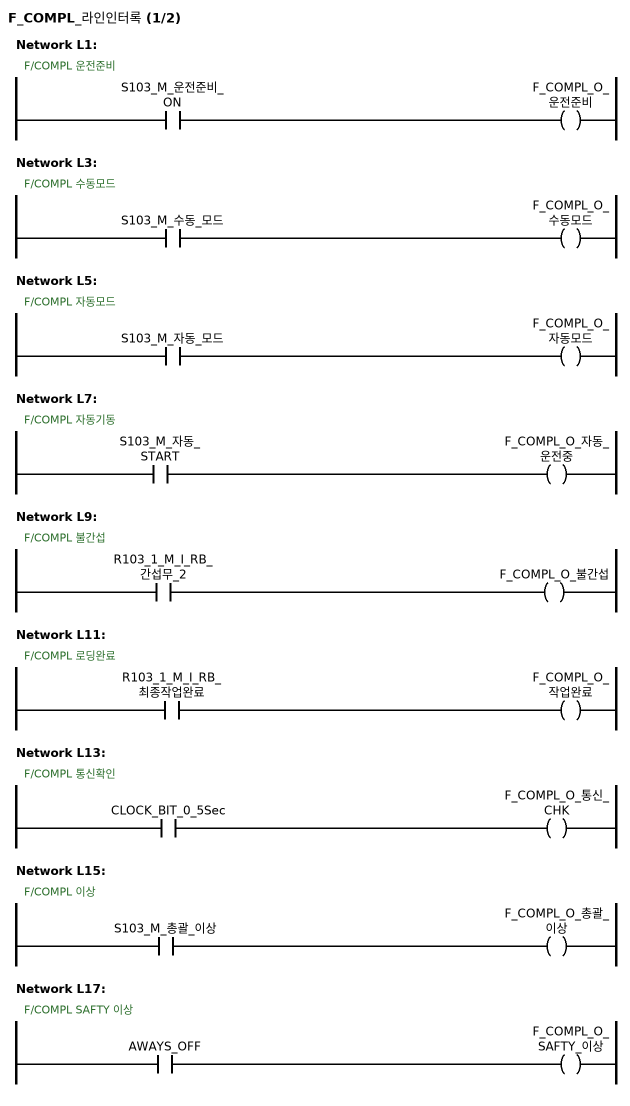
(* [picture p144: F_COMPL_라인인터록 rungs L1-L17] *)
(* F/COMPL 운전준비 *)
(* Rung L1 *)
F_COMPL_O_운전준비 := S103_M_운전준비_ON;
(* F/COMPL 수동모드 *)
(* Rung L3 *)
F_COMPL_O_수동모드 := S103_M_수동_모드;
(* F/COMPL 자동모드 *)
(* Rung L5 *)
F_COMPL_O_자동모드 := S103_M_자동_모드;
(* F/COMPL 자동기동 *)
(* Rung L7 *)
F_COMPL_O_자동_운전중 := S103_M_자동_START;
(* F/COMPL 불간섭 *)
(* Rung L9 *)
F_COMPL_O_불간섭 := R103_1_M_I_RB_간섭무_2;
(* F/COMPL 로딩완료 *)
(* Rung L11 *)
F_COMPL_O_작업완료 := R103_1_M_I_RB_최종작업완료;
(* F/COMPL 통신확인 *)
(* Rung L13 *)
F_COMPL_O_통신_CHK := CLOCK_BIT_0_5Sec;
(* F/COMPL 이상 *)
(* Rung L15 *)
F_COMPL_O_총괄_이상 := S103_M_총괄_이상;
(* F/COMPL SAFTY 이상 *)
(* Rung L17 *)
F_COMPL_O_SAFTY_이상 := AWAYS_OFF;

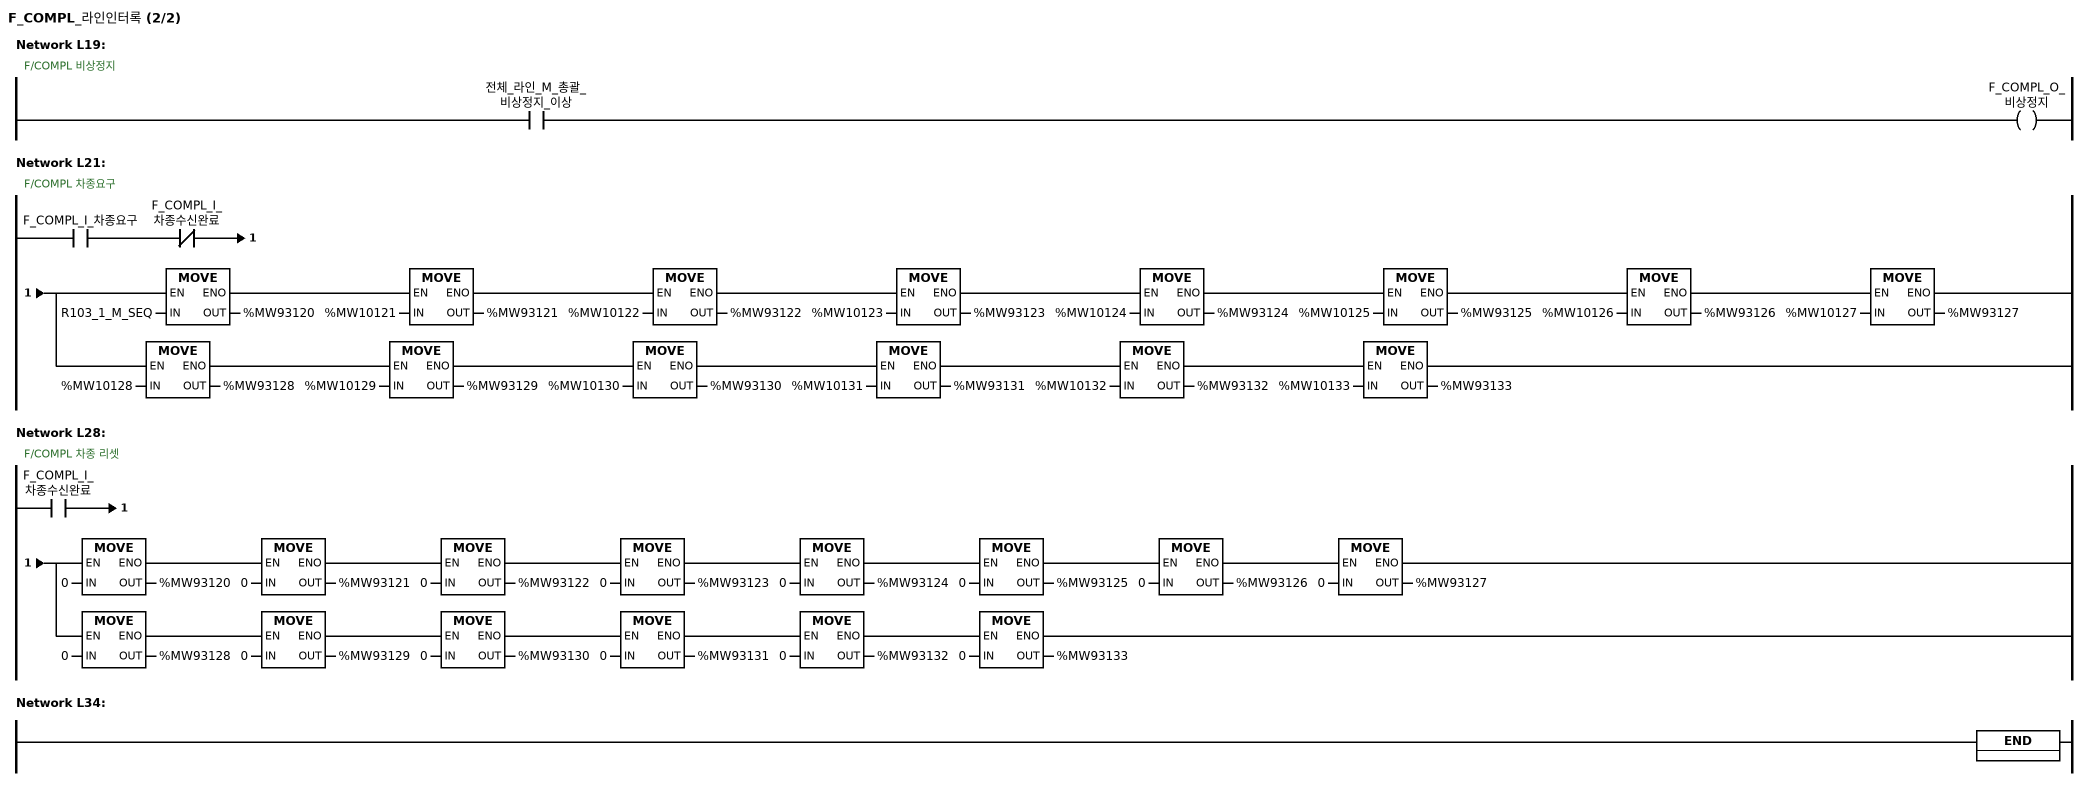
(* F/COMPL 비상정지 *)
(* Rung L19 *)
F_COMPL_O_비상정지 := 전체_라인_M_총괄_비상정지_이상;
(* F/COMPL 차종요구 *)
(* Rung L21 *)
IF F_COMPL_I_차종요구 AND NOT F_COMPL_I_차종수신완료 THEN
    %MW93120 := R103_1_M_SEQ;
    %MW93121 := %MW10121;
    %MW93122 := %MW10122;
    %MW93123 := %MW10123;
    %MW93124 := %MW10124;
    %MW93125 := %MW10125;
    %MW93126 := %MW10126;
    %MW93127 := %MW10127;
    %MW93128 := %MW10128;
    %MW93129 := %MW10129;
    %MW93130 := %MW10130;
    %MW93131 := %MW10131;
    %MW93132 := %MW10132;
    %MW93133 := %MW10133;
END_IF;
(* F/COMPL 차종 리셋 *)
(* Rung L28 *)
IF F_COMPL_I_차종수신완료 THEN
    %MW93120 := 0;
    %MW93121 := 0;
    %MW93122 := 0;
    %MW93123 := 0;
    %MW93124 := 0;
    %MW93125 := 0;
    %MW93126 := 0;
    %MW93127 := 0;
    %MW93128 := 0;
    %MW93129 := 0;
    %MW93130 := 0;
    %MW93131 := 0;
    %MW93132 := 0;
    %MW93133 := 0;
END_IF;
(* Rung L34 *)
END();
END_PROGRAM

PROGRAM 차종전송 (* task: 스캔 프로그램 *)
VAR_EXTERNAL
    AWAYS_OFF : BOOL; (* AT %MW3.0 *)
    AWAYS_ON : BOOL; (* AT %MW3.1 *)
    CARTYPE : ARRAY[0..999] OF WORD; (* AT %MW10000 *) (* CARTYPE *)
    F_COMPL_I_파트_ON : BOOL; (* AT %MW83210.8 *)
    R101_1_1_M_DATA_전송_MEMO : BOOL; (* AT %MW9000.8 *) (* R101_1_1_M_DATA_전송_MEMO *)
    R101_1_1_M_DATA_전송_PLS : BOOL; (* AT %MW9000.9 *) (* R101_1_1_M_DATA_전송_PLS *)
    R101_1_1_M_DATA_전송_완료 : BOOL; (* AT %MW9000.11 *) (* R101_1_1_M_DATA_전송_완료 *)
    R101_1_1_M_STN_차종_ON : BOOL; (* AT %MW1002.2 *)
    R101_1_M_I_RB_2차_작업완료 : BOOL; (* AT %MW20071.3 *)
    R101_1_M_I_RB_원위치 : BOOL; (* AT %MW20070.3 *)
    R101_1_S101_CTYPE_MOVE : FB407_Car_Type_Move_Stn_v1;
    R101_1_S102_CTYPE_MOVE : FB407_Car_Type_Move_Stn_v1;
    R102_1_1_M_DATA_삭제_PLS : BOOL; (* AT %MW9002.0 *) (* R102_1_1_M_DATA_삭제_PLS *)
    R102_1_1_M_DATA_삭제_완료 : BOOL; (* AT %MW9002.2 *) (* R102_1_1_M_DATA_삭제_완료 *)
    R102_1_1_M_DATA_전송_MEMO : BOOL; (* AT %MW9002.8 *) (* R102_1_1_M_DATA_전송_MEMO *)
    R102_1_1_M_DATA_전송_PLS : BOOL; (* AT %MW9002.9 *) (* R102_1_1_M_DATA_전송_PLS *)
    R102_1_1_M_DATA_전송_완료 : BOOL; (* AT %MW9002.11 *) (* R102_1_1_M_DATA_전송_완료 *)
    R102_1_1_M_I_RB_2차_작업완료 : BOOL; (* AT %MW20091.3 *)
    R102_1_1_M_I_RB_원위치 : BOOL; (* AT %MW20090.3 *)
    R102_1_1_M_STN_차종_ON : BOOL; (* AT %MW1502.2 *)
    R102_1_1_S102_CTYPE_MOVE : FB407_Car_Type_Move_Stn_v1;
    R102_1_1_S103_CTYPE_MOVE : FB407_Car_Type_Move_Stn_v1;
    R102_1_CTYPE_CLEAR : FB409_Car_Type_Clear_v1;
    R102_1_M_DATA_전송_MEMO : BOOL; (* AT %MW9004.8 *) (* R102_1_M_DATA_전송_MEMO *)
    R102_1_M_DATA_전송_PLS : BOOL; (* AT %MW9004.9 *) (* R102_1_M_DATA_전송_PLS *)
    R102_1_M_DATA_전송_완료 : BOOL; (* AT %MW9004.11 *) (* R102_1_M_DATA_전송_완료 *)
    R102_1_M_I_RB_1차_작업완료 : BOOL; (* AT %MW20081.2 *)
    R102_1_M_I_RB_2차_작업완료 : BOOL; (* AT %MW20081.3 *)
    R102_1_M_I_RB_원위치 : BOOL; (* AT %MW20080.3 *)
    R102_1_M_STN_차종_NONE : BOOL; (* AT %MW1502.5 *)
    R102_1_M_STN_차종_ON : BOOL; (* AT %MW1502.4 *)
    R102_1_S103_CTYPE_MOVE : FB407_Car_Type_Move_Stn_v1;
    R102_1_S104_CTYPE_MOVE : FB407_Car_Type_Move_Stn_v1;
    R102_2_CTYPE_CLEAR : FB409_Car_Type_Clear_v1;
    R103_1_M_DATA_삭제_PLS : BOOL; (* AT %MW9006.0 *) (* R103_1_M_DATA_삭제_PLS *)
    R103_1_M_DATA_삭제_완료 : BOOL; (* AT %MW9006.2 *) (* R103_1_M_DATA_삭제_완료 *)
    R103_1_M_I_RB_1차_작업완료 : BOOL; (* AT %MW20101.2 *)
    R103_1_M_I_RB_2차_작업완료 : BOOL; (* AT %MW20101.3 *)
    R103_1_M_STN_차종_NONE : BOOL; (* AT %MW2002.3 *)
    S101_M_DATA_전송_MEMO : BOOL; (* AT %MW9001.8 *) (* S101_M_DATA_전송_MEMO *)
    S101_M_DATA_전송_PLS : BOOL; (* AT %MW9001.9 *) (* S101_M_DATA_전송_PLS *)
    S101_M_DATA_전송_완료 : BOOL; (* AT %MW9001.11 *) (* S101_M_DATA_전송_완료 *)
    S101_M_STN_DASH_로딩완료 : BOOL; (* AT %MW1001.12 *)
    S101_M_STN_LH_로딩완료 : BOOL; (* AT %MW1001.10 *)
    S101_M_STN_RH_로딩완료 : BOOL; (* AT %MW1001.11 *)
    S101_M_STN_차종_NONE : BOOL; (* AT %MW1002.1 *)
    S101_M_STN_차종_ON : BOOL; (* AT %MW1002.0 *)
    S101_M_공정_APRON_제품감지_OFF : BOOL; (* AT %MW1001.4 *)
    S101_M_공정_APRON_제품감지_ON : BOOL; (* AT %MW1001.3 *)
    S101_M_공정_DASH_제품감지_OFF : BOOL; (* AT %MW1001.6 *)
    S101_M_작업_완료 : BOOL; (* AT %MW1001.0 *)
    S101_R102_2_CTYPE_MOVE : FB407_Car_Type_Move_Stn_v1;
    S101_R102_3_CTYPE_MOVE : FB407_Car_Type_Move_Stn_v1;
    S102_M_DATA_전송_MEMO : BOOL; (* AT %MW9003.8 *) (* S102_M_DATA_전송_MEMO *)
    S102_M_DATA_전송_PLS : BOOL; (* AT %MW9003.9 *) (* S102_M_DATA_전송_PLS *)
    S102_M_DATA_전송_완료 : BOOL; (* AT %MW9003.11 *) (* S102_M_DATA_전송_완료 *)
    S102_M_STN_DASH_로딩완료 : BOOL; (* AT %MW1501.8 *)
    S102_M_STN_차종_NONE : BOOL; (* AT %MW1502.1 *)
    S102_M_STN_차종_ON : BOOL; (* AT %MW1502.0 *)
    S102_M_공정_제품감지_OFF : BOOL; (* AT %MW1501.4 *)
    S102_M_공정_제품감지_ON : BOOL; (* AT %MW1501.3 *)
    S102_M_작업_완료 : BOOL; (* AT %MW1501.0 *)
    S102_R102_1_CTYPE_MOVE : FB407_Car_Type_Move_Stn_v1;
    S102_R102_2_CTYPE_MOVE : FB407_Car_Type_Move_Stn_v1;
    S103_M_DATA_전송_MEMO : BOOL; (* AT %MW9005.8 *) (* S103_M_DATA_전송_MEMO *)
    S103_M_DATA_전송_PLS : BOOL; (* AT %MW9005.9 *) (* S103_M_DATA_전송_PLS *)
    S103_M_DATA_전송_완료 : BOOL; (* AT %MW9005.11 *) (* S103_M_DATA_전송_완료 *)
    S103_M_STN_FRT_FLR_로딩완료 : BOOL; (* AT %MW2001.8 *)
    S103_M_STN_차종_NONE : BOOL; (* AT %MW2002.1 *)
    S103_M_STN_차종_ON : BOOL; (* AT %MW2002.0 *)
    S103_M_공정_제품감지_OFF : BOOL; (* AT %MW2001.4 *)
    S103_M_공정_제품감지_ON : BOOL; (* AT %MW2001.3 *)
    S103_M_작업_완료 : BOOL; (* AT %MW2001.0 *)
    S103_R103_1_CTYPE_MOVE : FB407_Car_Type_Move_Stn_v1;
    S103_R103_2_CTYPE_MOVE : FB407_Car_Type_Move_Stn_v1;
END_VAR
VAR
    _e1 : R_TRIG;
    _e2 : R_TRIG;
    _e3 : R_TRIG;
    _e4 : R_TRIG;
    _e5 : R_TRIG;
    _e6 : R_TRIG;
END_VAR

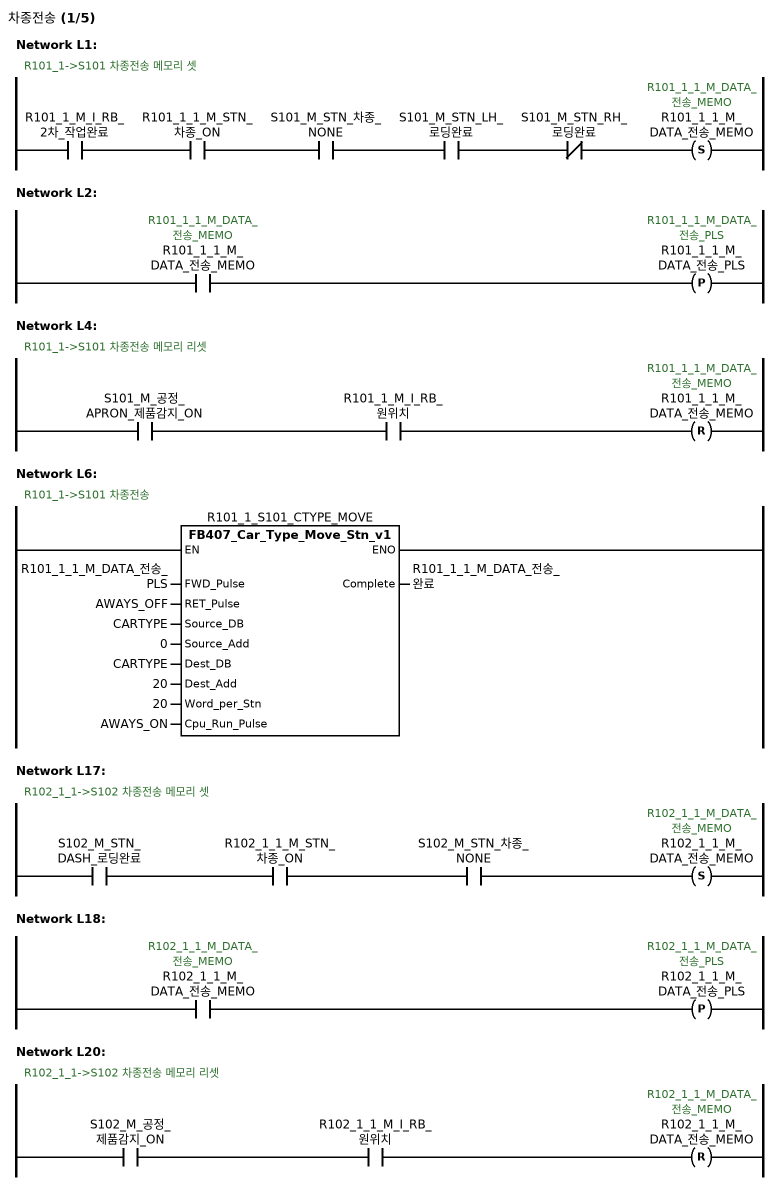
(* R101_1->S101 차종전송 메모리 셋 *)
(* Rung L1 *)
IF R101_1_M_I_RB_2차_작업완료 AND R101_1_1_M_STN_차종_ON AND S101_M_STN_차종_NONE AND S101_M_STN_LH_로딩완료 AND NOT S101_M_STN_RH_로딩완료 THEN
    R101_1_1_M_DATA_전송_MEMO := TRUE;
END_IF;
(* Rung L2 *)
_e1(CLK := R101_1_1_M_DATA_전송_MEMO);
R101_1_1_M_DATA_전송_PLS := _e1.Q;
(* R101_1->S101 차종전송 메모리 리셋 *)
(* Rung L4 *)
IF S101_M_공정_APRON_제품감지_ON AND R101_1_M_I_RB_원위치 THEN R101_1_1_M_DATA_전송_MEMO := FALSE; END_IF;
(* R101_1->S101 차종전송 *)
(* Rung L6 *)
R101_1_S101_CTYPE_MOVE(FWD_Pulse := R101_1_1_M_DATA_전송_PLS, RET_Pulse := AWAYS_OFF, Source_DB := CARTYPE, Source_Add := 0, Dest_DB := CARTYPE, Dest_Add := 20, Word_per_Stn := 20, Cpu_Run_Pulse := AWAYS_ON, Complete => R101_1_1_M_DATA_전송_완료);
(* R102_1_1->S102 차종전송 메모리 셋 *)
(* Rung L17 *)
IF S102_M_STN_DASH_로딩완료 AND R102_1_1_M_STN_차종_ON AND S102_M_STN_차종_NONE THEN
    R102_1_1_M_DATA_전송_MEMO := TRUE;
END_IF;
(* Rung L18 *)
_e2(CLK := R102_1_1_M_DATA_전송_MEMO);
R102_1_1_M_DATA_전송_PLS := _e2.Q;
(* R102_1_1->S102 차종전송 메모리 리셋 *)
(* Rung L20 *)
IF S102_M_공정_제품감지_ON AND R102_1_1_M_I_RB_원위치 THEN R102_1_1_M_DATA_전송_MEMO := FALSE; END_IF;

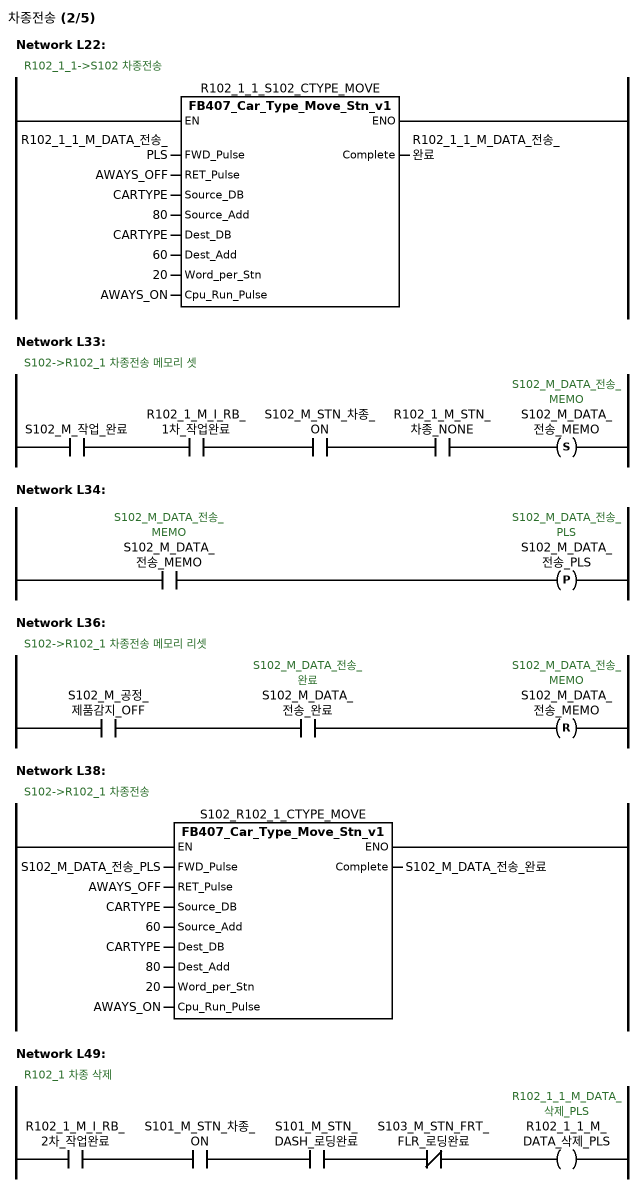
(* R102_1_1->S102 차종전송 *)
(* Rung L22 *)
R102_1_1_S102_CTYPE_MOVE(FWD_Pulse := R102_1_1_M_DATA_전송_PLS, RET_Pulse := AWAYS_OFF, Source_DB := CARTYPE, Source_Add := 80, Dest_DB := CARTYPE, Dest_Add := 60, Word_per_Stn := 20, Cpu_Run_Pulse := AWAYS_ON, Complete => R102_1_1_M_DATA_전송_완료);
(* S102->R102_1 차종전송 메모리 셋 *)
(* Rung L33 *)
IF S102_M_작업_완료 AND R102_1_M_I_RB_1차_작업완료 AND S102_M_STN_차종_ON AND R102_1_M_STN_차종_NONE THEN
    S102_M_DATA_전송_MEMO := TRUE;
END_IF;
(* Rung L34 *)
_e3(CLK := S102_M_DATA_전송_MEMO);
S102_M_DATA_전송_PLS := _e3.Q;
(* S102->R102_1 차종전송 메모리 리셋 *)
(* Rung L36 *)
IF S102_M_공정_제품감지_OFF AND S102_M_DATA_전송_완료 THEN S102_M_DATA_전송_MEMO := FALSE; END_IF;
(* S102->R102_1 차종전송 *)
(* Rung L38 *)
S102_R102_1_CTYPE_MOVE(FWD_Pulse := S102_M_DATA_전송_PLS, RET_Pulse := AWAYS_OFF, Source_DB := CARTYPE, Source_Add := 60, Dest_DB := CARTYPE, Dest_Add := 80, Word_per_Stn := 20, Cpu_Run_Pulse := AWAYS_ON, Complete => S102_M_DATA_전송_완료);
(* R102_1 차종 삭제 *)
(* Rung L49 *)
R102_1_1_M_DATA_삭제_PLS := R102_1_M_I_RB_2차_작업완료 AND S101_M_STN_차종_ON AND S101_M_STN_DASH_로딩완료 AND NOT S103_M_STN_FRT_FLR_로딩완료;

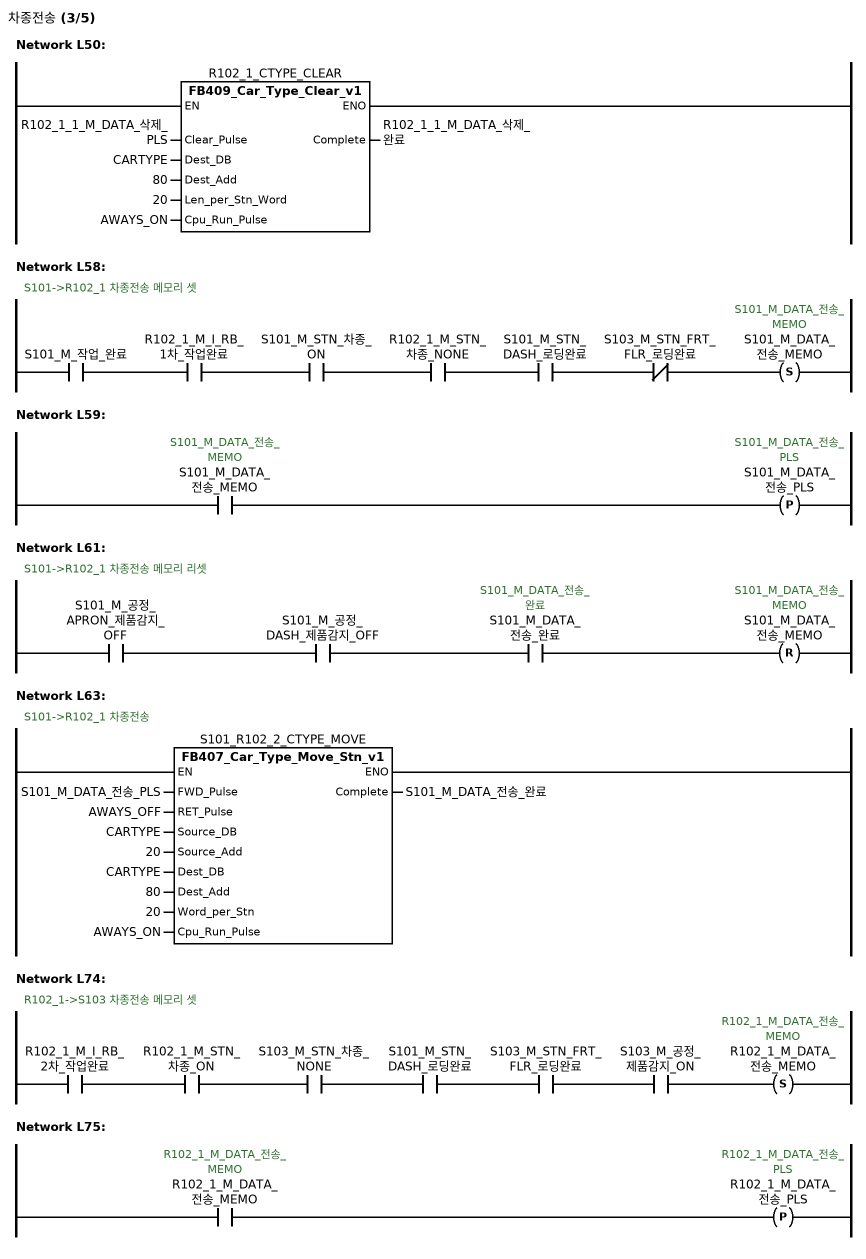
(* Rung L50 *)
R102_1_CTYPE_CLEAR(Clear_Pulse := R102_1_1_M_DATA_삭제_PLS, Dest_DB := CARTYPE, Dest_Add := 80, Len_per_Stn_Word := 20, Cpu_Run_Pulse := AWAYS_ON, Complete => R102_1_1_M_DATA_삭제_완료);
(* S101->R102_1 차종전송 메모리 셋 *)
(* Rung L58 *)
IF S101_M_작업_완료 AND R102_1_M_I_RB_1차_작업완료 AND S101_M_STN_차종_ON AND R102_1_M_STN_차종_NONE AND S101_M_STN_DASH_로딩완료 AND NOT S103_M_STN_FRT_FLR_로딩완료 THEN
    S101_M_DATA_전송_MEMO := TRUE;
END_IF;
(* Rung L59 *)
_e4(CLK := S101_M_DATA_전송_MEMO);
S101_M_DATA_전송_PLS := _e4.Q;
(* S101->R102_1 차종전송 메모리 리셋 *)
(* Rung L61 *)
IF S101_M_공정_APRON_제품감지_OFF AND S101_M_공정_DASH_제품감지_OFF AND S101_M_DATA_전송_완료 THEN
    S101_M_DATA_전송_MEMO := FALSE;
END_IF;
(* S101->R102_1 차종전송 *)
(* Rung L63 *)
S101_R102_2_CTYPE_MOVE(FWD_Pulse := S101_M_DATA_전송_PLS, RET_Pulse := AWAYS_OFF, Source_DB := CARTYPE, Source_Add := 20, Dest_DB := CARTYPE, Dest_Add := 80, Word_per_Stn := 20, Cpu_Run_Pulse := AWAYS_ON, Complete => S101_M_DATA_전송_완료);
(* R102_1->S103 차종전송 메모리 셋 *)
(* Rung L74 *)
IF R102_1_M_I_RB_2차_작업완료 AND R102_1_M_STN_차종_ON AND S103_M_STN_차종_NONE AND S101_M_STN_DASH_로딩완료 AND S103_M_STN_FRT_FLR_로딩완료 AND S103_M_공정_제품감지_ON THEN
    R102_1_M_DATA_전송_MEMO := TRUE;
END_IF;
(* Rung L75 *)
_e5(CLK := R102_1_M_DATA_전송_MEMO);
R102_1_M_DATA_전송_PLS := _e5.Q;

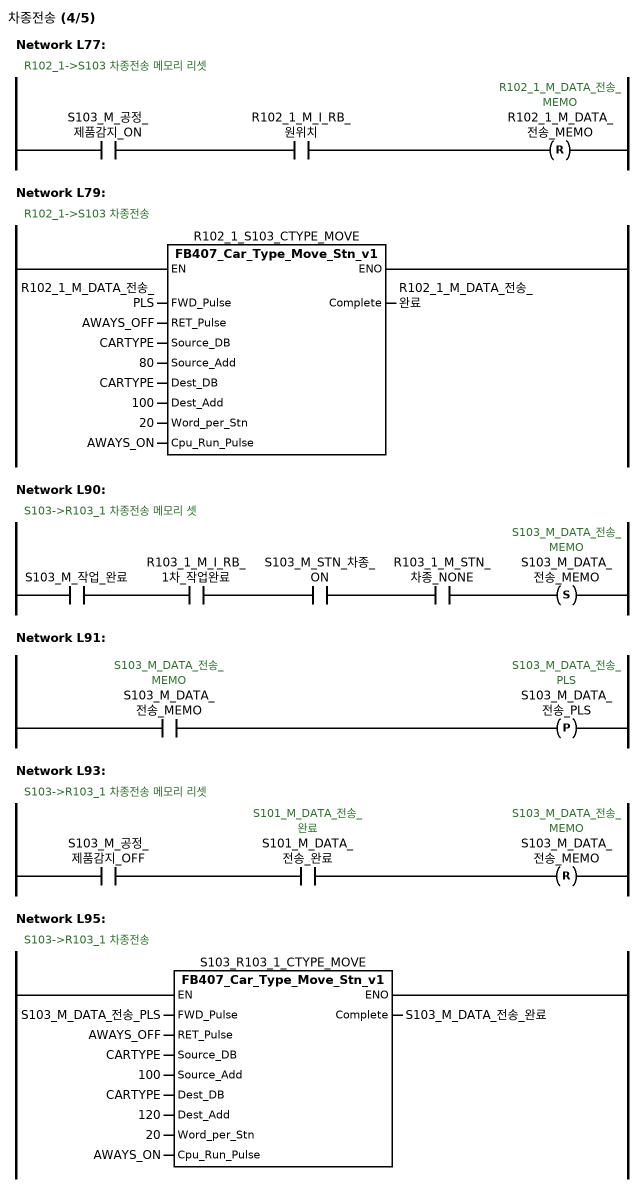
(* R102_1->S103 차종전송 메모리 리셋 *)
(* Rung L77 *)
IF S103_M_공정_제품감지_ON AND R102_1_M_I_RB_원위치 THEN R102_1_M_DATA_전송_MEMO := FALSE; END_IF;
(* R102_1->S103 차종전송 *)
(* Rung L79 *)
R102_1_S103_CTYPE_MOVE(FWD_Pulse := R102_1_M_DATA_전송_PLS, RET_Pulse := AWAYS_OFF, Source_DB := CARTYPE, Source_Add := 80, Dest_DB := CARTYPE, Dest_Add := 100, Word_per_Stn := 20, Cpu_Run_Pulse := AWAYS_ON, Complete => R102_1_M_DATA_전송_완료);
(* S103->R103_1 차종전송 메모리 셋 *)
(* Rung L90 *)
IF S103_M_작업_완료 AND R103_1_M_I_RB_1차_작업완료 AND S103_M_STN_차종_ON AND R103_1_M_STN_차종_NONE THEN
    S103_M_DATA_전송_MEMO := TRUE;
END_IF;
(* Rung L91 *)
_e6(CLK := S103_M_DATA_전송_MEMO);
S103_M_DATA_전송_PLS := _e6.Q;
(* S103->R103_1 차종전송 메모리 리셋 *)
(* Rung L93 *)
IF S103_M_공정_제품감지_OFF AND S101_M_DATA_전송_완료 THEN S103_M_DATA_전송_MEMO := FALSE; END_IF;
(* S103->R103_1 차종전송 *)
(* Rung L95 *)
S103_R103_1_CTYPE_MOVE(FWD_Pulse := S103_M_DATA_전송_PLS, RET_Pulse := AWAYS_OFF, Source_DB := CARTYPE, Source_Add := 100, Dest_DB := CARTYPE, Dest_Add := 120, Word_per_Stn := 20, Cpu_Run_Pulse := AWAYS_ON, Complete => S103_M_DATA_전송_완료);

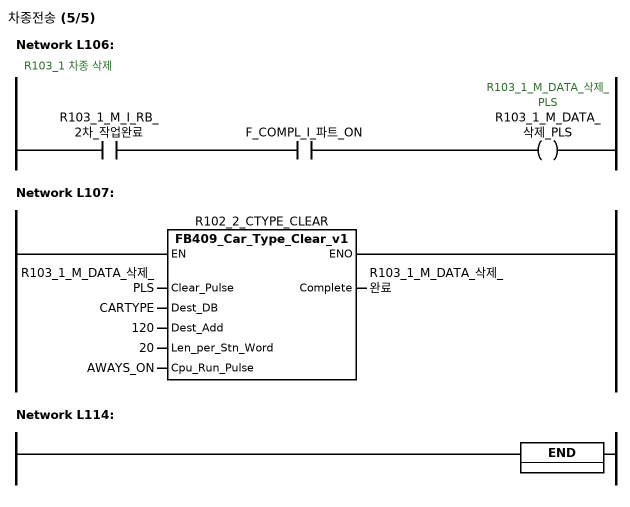
(* R103_1 차종 삭제 *)
(* Rung L106 *)
R103_1_M_DATA_삭제_PLS := R103_1_M_I_RB_2차_작업완료 AND F_COMPL_I_파트_ON;
(* Rung L107 *)
R102_2_CTYPE_CLEAR(Clear_Pulse := R103_1_M_DATA_삭제_PLS, Dest_DB := CARTYPE, Dest_Add := 120, Len_per_Stn_Word := 20, Cpu_Run_Pulse := AWAYS_ON, Complete => R103_1_M_DATA_삭제_완료);
(* Rung L114 *)
END();
END_PROGRAM

PROGRAM HMI_차종수정 (* task: 스캔 프로그램 *)
VAR_EXTERNAL
    CARTYPE : ARRAY[0..999] OF WORD; (* AT %MW10000 *) (* CARTYPE *)
    HMI_M_매칭_R102_1_S101 : BOOL; (* AT %MW70.1 *)
    HMI_M_매칭_S101_R102_1 : BOOL; (* AT %MW70.0 *)
    HMI_M_매칭선택 : WORD; (* AT %MW70 *)
    HMI_M_매칭차종_DATA_OK : BOOL; (* AT %MW9.9 *)
    HMI_M_매칭차종_복사_ON : BOOL; (* AT %MW9.6 *)
    HMI_M_매칭차종_복사_SET : BOOL; (* AT %MW9.8 *)
    HMI_M_차종매칭_SEQ : WORD; (* AT %MW50 *)
    HMI_M_차종매칭_차종1_AX : BOOL; (* AT %MW51.0 *)
    HMI_M_차종매칭_차종1_B : BOOL; (* AT %MW51.1 *)
    HMI_M_차종매칭_차종1_C : BOOL; (* AT %MW51.2 *)
    HMI_M_차종매칭_차종1_D : BOOL; (* AT %MW51.3 *)
    HMI_M_차종매칭_차종1_E : BOOL; (* AT %MW51.4 *)
    HMI_M_차종매칭_차종1_F : BOOL; (* AT %MW51.5 *)
    HMI_M_차종매칭_차종1_G : BOOL; (* AT %MW51.6 *)
    HMI_M_차종매칭_차종1_H : BOOL; (* AT %MW51.7 *)
    HMI_M_차종매칭_차종2_3DR : BOOL; (* AT %MW51.8 *)
    HMI_M_차종매칭_차종2_4DR : BOOL; (* AT %MW51.9 *)
    HMI_M_차종매칭_차종2_5DR : BOOL; (* AT %MW51.10 *)
    HMI_M_차종매칭_차종2_SP1 : BOOL; (* AT %MW51.12 *)
    HMI_M_차종매칭_차종2_SP2 : BOOL; (* AT %MW51.13 *)
    HMI_M_차종매칭_차종2_WGN : BOOL; (* AT %MW51.11 *)
    HMI_M_차종매칭_차종3_LHD : BOOL; (* AT %MW51.14 *)
    HMI_M_차종매칭_차종3_RHD : BOOL; (* AT %MW51.15 *)
    HMI_M_차종매칭_차종4_EEC : BOOL; (* AT %MW52.3 *)
    HMI_M_차종매칭_차종4_SP1 : BOOL; (* AT %MW52.8 *)
    HMI_M_차종매칭_차종4_SP2 : BOOL; (* AT %MW52.9 *)
    HMI_M_차종매칭_차종4_SP3 : BOOL; (* AT %MW52.11 *)
    HMI_M_차종매칭_차종4_SP4 : BOOL; (* AT %MW52.12 *)
    HMI_M_차종매칭_차종4_SP5 : BOOL; (* AT %MW52.13 *)
    HMI_M_차종매칭_차종4_SP6 : BOOL; (* AT %MW52.14 *)
    HMI_M_차종매칭_차종4_SP7 : BOOL; (* AT %MW52.15 *)
    HMI_M_차종매칭_차종4_내수 : BOOL; (* AT %MW52.0 *)
    HMI_M_차종매칭_차종4_러시아 : BOOL; (* AT %MW52.10 *)
    HMI_M_차종매칭_차종4_북미 : BOOL; (* AT %MW52.2 *)
    HMI_M_차종매칭_차종4_브라질 : BOOL; (* AT %MW52.7 *)
    HMI_M_차종매칭_차종4_수출 : BOOL; (* AT %MW52.1 *)
    HMI_M_차종매칭_차종4_중국 : BOOL; (* AT %MW52.6 *)
    HMI_M_차종매칭_차종4_중동 : BOOL; (* AT %MW52.5 *)
    HMI_M_차종매칭_차종4_호주 : BOOL; (* AT %MW52.4 *)
    HMI_M_차종매칭_차종5_AT : BOOL; (* AT %MW53.1 *)
    HMI_M_차종매칭_차종5_MT : BOOL; (* AT %MW53.0 *)
    HMI_M_차종매칭_차종5_SP1 : BOOL; (* AT %MW53.2 *)
    HMI_M_차종매칭_차종6_DSROOF : BOOL; (* AT %MW53.6 *)
    HMI_M_차종매칭_차종6_SP1 : BOOL; (* AT %MW53.7 *)
    HMI_M_차종매칭_차종6_썬루프 : BOOL; (* AT %MW53.4 *)
    HMI_M_차종매칭_차종6_일반루프 : BOOL; (* AT %MW53.3 *)
    HMI_M_차종매칭_차종6_파노라마루프 : BOOL; (* AT %MW53.5 *)
    HMI_M_차종매칭_차종7_DSL : BOOL; (* AT %MW53.9 *)
    HMI_M_차종매칭_차종7_GSL : BOOL; (* AT %MW53.8 *)
    HMI_M_차종매칭_차종7_SP1 : BOOL; (* AT %MW53.10 *)
    HMI_M_차종매칭_차종7_SP2 : BOOL; (* AT %MW53.11 *)
    HMI_M_차종매칭_차종7_SP3 : BOOL; (* AT %MW53.12 *)
    HMI_M_차종매칭_차종7_SP4 : BOOL; (* AT %MW53.13 *)
    HMI_M_차종매칭_차종7_SP5 : BOOL; (* AT %MW53.14 *)
    HMI_M_차종매칭_차종7_SP6 : BOOL; (* AT %MW53.15 *)
    HMI_M_차종매칭_차종8_2WD : BOOL; (* AT %MW54.0 *)
    HMI_M_차종매칭_차종8_4WD : BOOL; (* AT %MW54.1 *)
    HMI_M_차종매칭_차종8_SP1 : BOOL; (* AT %MW54.2 *)
    HMI_M_차종매칭_차종9_MPI : BOOL; (* AT %MW54.3 *)
    HMI_M_차종매칭_차종9_SP1 : BOOL; (* AT %MW54.5 *)
    HMI_M_차종매칭_차종9_SP10 : BOOL; (* AT %MW54.14 *)
    HMI_M_차종매칭_차종9_SP11 : BOOL; (* AT %MW54.15 *)
    HMI_M_차종매칭_차종9_SP2 : BOOL; (* AT %MW54.6 *)
    HMI_M_차종매칭_차종9_SP3 : BOOL; (* AT %MW54.7 *)
    HMI_M_차종매칭_차종9_SP4 : BOOL; (* AT %MW54.8 *)
    HMI_M_차종매칭_차종9_SP5 : BOOL; (* AT %MW54.9 *)
    HMI_M_차종매칭_차종9_SP6 : BOOL; (* AT %MW54.10 *)
    HMI_M_차종매칭_차종9_SP7 : BOOL; (* AT %MW54.11 *)
    HMI_M_차종매칭_차종9_SP8 : BOOL; (* AT %MW54.12 *)
    HMI_M_차종매칭_차종9_SP9 : BOOL; (* AT %MW54.13 *)
    HMI_M_차종매칭_차종9_T_GDI : BOOL; (* AT %MW54.4 *)
    HMI_M_차종매칭_차종_OPT1_R_RACK_무 : BOOL; (* AT %MW55.3 *)
    HMI_M_차종매칭_차종_OPT1_R_RACK_유 : BOOL; (* AT %MW55.2 *)
    HMI_M_차종매칭_차종_OPT1_S_REP_EATER_무 : BOOL; (* AT %MW55.7 *)
    HMI_M_차종매칭_차종_OPT1_S_REP_EATER_유 : BOOL; (* AT %MW55.6 *)
    HMI_M_차종매칭_차종_OPT1_VAN_무 : BOOL; (* AT %MW55.9 *)
    HMI_M_차종매칭_차종_OPT1_VAN_유 : BOOL; (* AT %MW55.8 *)
    HMI_M_차종매칭_차종_OPT1_슬라이딩_무 : BOOL; (* AT %MW55.1 *)
    HMI_M_차종매칭_차종_OPT1_슬라이딩_유 : BOOL; (* AT %MW55.0 *)
    HMI_M_차종매칭_차종_OPT1_폴딩_무 : BOOL; (* AT %MW55.5 *)
    HMI_M_차종매칭_차종_OPT1_폴딩_유 : BOOL; (* AT %MW55.4 *)
    HMI_M_차종매칭_차종_공대차 : BOOL; (* AT %MW60.12 *)
    HMI_M_차종매칭_차종_공차 : BOOL; (* AT %MW60.10 *)
    HMI_M_차종매칭_차종_불량대차 : BOOL; (* AT %MW60.13 *)
    HMI_M_차종매칭_차종_불량차 : BOOL; (* AT %MW60.11 *)
    HMI_M_차종수정 : ARRAY[0..19] OF WORD; (* AT %MW10 *)
    HMI_M_차종수정_DATA_OK : BOOL; (* AT %MW9.0 *)
    HMI_M_차종수정_RESET : BOOL; (* AT %MW9.2 *)
    HMI_M_차종수정_SEQ : WORD; (* AT %MW10 *)
    HMI_M_차종수정_SET : BOOL; (* AT %MW9.1 *)
    HMI_M_차종수정_차종1_AX : BOOL; (* AT %MW11.0 *)
    HMI_M_차종수정_차종1_B : BOOL; (* AT %MW11.1 *)
    HMI_M_차종수정_차종1_C : BOOL; (* AT %MW11.2 *)
    HMI_M_차종수정_차종1_D : BOOL; (* AT %MW11.3 *)
    HMI_M_차종수정_차종1_E : BOOL; (* AT %MW11.4 *)
    HMI_M_차종수정_차종1_F : BOOL; (* AT %MW11.5 *)
    HMI_M_차종수정_차종1_G : BOOL; (* AT %MW11.6 *)
    HMI_M_차종수정_차종1_H : BOOL; (* AT %MW11.7 *)
    HMI_M_차종수정_차종2_3DR : BOOL; (* AT %MW11.8 *)
    HMI_M_차종수정_차종2_4DR : BOOL; (* AT %MW11.9 *)
    HMI_M_차종수정_차종2_5DR : BOOL; (* AT %MW11.10 *)
    HMI_M_차종수정_차종2_SP1 : BOOL; (* AT %MW11.12 *)
    HMI_M_차종수정_차종2_SP2 : BOOL; (* AT %MW11.13 *)
    HMI_M_차종수정_차종2_WGN : BOOL; (* AT %MW11.11 *)
    HMI_M_차종수정_차종3_LHD : BOOL; (* AT %MW11.14 *)
    HMI_M_차종수정_차종3_RHD : BOOL; (* AT %MW11.15 *)
    HMI_M_차종수정_차종4_EEC : BOOL; (* AT %MW12.3 *)
    HMI_M_차종수정_차종4_SP1 : BOOL; (* AT %MW12.8 *)
    HMI_M_차종수정_차종4_SP2 : BOOL; (* AT %MW12.9 *)
    HMI_M_차종수정_차종4_SP3 : BOOL; (* AT %MW12.11 *)
    HMI_M_차종수정_차종4_SP4 : BOOL; (* AT %MW12.12 *)
    HMI_M_차종수정_차종4_SP5 : BOOL; (* AT %MW12.13 *)
    HMI_M_차종수정_차종4_SP6 : BOOL; (* AT %MW12.14 *)
    HMI_M_차종수정_차종4_SP7 : BOOL; (* AT %MW12.15 *)
    HMI_M_차종수정_차종4_내수 : BOOL; (* AT %MW12.0 *)
    HMI_M_차종수정_차종4_러시아 : BOOL; (* AT %MW12.10 *)
    HMI_M_차종수정_차종4_북미 : BOOL; (* AT %MW12.2 *)
    HMI_M_차종수정_차종4_브라질 : BOOL; (* AT %MW12.7 *)
    HMI_M_차종수정_차종4_수출 : BOOL; (* AT %MW12.1 *)
    HMI_M_차종수정_차종4_중국 : BOOL; (* AT %MW12.6 *)
    HMI_M_차종수정_차종4_중동 : BOOL; (* AT %MW12.5 *)
    HMI_M_차종수정_차종4_호주 : BOOL; (* AT %MW12.4 *)
    HMI_M_차종수정_차종5_AT : BOOL; (* AT %MW13.1 *)
    HMI_M_차종수정_차종5_MT : BOOL; (* AT %MW13.0 *)
    HMI_M_차종수정_차종5_SP1 : BOOL; (* AT %MW13.2 *)
    HMI_M_차종수정_차종6_DSROOF : BOOL; (* AT %MW13.6 *)
    HMI_M_차종수정_차종6_SP1 : BOOL; (* AT %MW13.7 *)
    HMI_M_차종수정_차종6_썬루프 : BOOL; (* AT %MW13.4 *)
    HMI_M_차종수정_차종6_일반루프 : BOOL; (* AT %MW13.3 *)
    HMI_M_차종수정_차종6_파노라마루프 : BOOL; (* AT %MW13.5 *)
    HMI_M_차종수정_차종7_DSL : BOOL; (* AT %MW13.9 *)
    HMI_M_차종수정_차종7_GSL : BOOL; (* AT %MW13.8 *)
    HMI_M_차종수정_차종7_SP1 : BOOL; (* AT %MW13.10 *)
    HMI_M_차종수정_차종7_SP2 : BOOL; (* AT %MW13.11 *)
    HMI_M_차종수정_차종7_SP3 : BOOL; (* AT %MW13.12 *)
    HMI_M_차종수정_차종7_SP4 : BOOL; (* AT %MW13.13 *)
    HMI_M_차종수정_차종7_SP5 : BOOL; (* AT %MW13.14 *)
    HMI_M_차종수정_차종7_SP6 : BOOL; (* AT %MW13.15 *)
    HMI_M_차종수정_차종8_2WD : BOOL; (* AT %MW14.0 *)
    HMI_M_차종수정_차종8_4WD : BOOL; (* AT %MW14.1 *)
    HMI_M_차종수정_차종8_SP1 : BOOL; (* AT %MW14.2 *)
    HMI_M_차종수정_차종9_MPI : BOOL; (* AT %MW14.3 *)
    HMI_M_차종수정_차종9_SP1 : BOOL; (* AT %MW14.5 *)
    HMI_M_차종수정_차종9_SP10 : BOOL; (* AT %MW14.14 *)
    HMI_M_차종수정_차종9_SP11 : BOOL; (* AT %MW14.15 *)
    HMI_M_차종수정_차종9_SP2 : BOOL; (* AT %MW14.6 *)
    HMI_M_차종수정_차종9_SP3 : BOOL; (* AT %MW14.7 *)
    HMI_M_차종수정_차종9_SP4 : BOOL; (* AT %MW14.8 *)
    HMI_M_차종수정_차종9_SP5 : BOOL; (* AT %MW14.9 *)
    HMI_M_차종수정_차종9_SP6 : BOOL; (* AT %MW14.10 *)
    HMI_M_차종수정_차종9_SP7 : BOOL; (* AT %MW14.11 *)
    HMI_M_차종수정_차종9_SP8 : BOOL; (* AT %MW14.12 *)
    HMI_M_차종수정_차종9_SP9 : BOOL; (* AT %MW14.13 *)
    HMI_M_차종수정_차종9_T_GDI : BOOL; (* AT %MW14.4 *)
    HMI_M_차종수정_차종_OPT1_R_RACK_무 : BOOL; (* AT %MW15.3 *)
    HMI_M_차종수정_차종_OPT1_R_RACK_유 : BOOL; (* AT %MW15.2 *)
    HMI_M_차종수정_차종_OPT1_S_REP_EATER_무 : BOOL; (* AT %MW15.7 *)
    HMI_M_차종수정_차종_OPT1_S_REP_EATER_유 : BOOL; (* AT %MW15.6 *)
    HMI_M_차종수정_차종_OPT1_VAN_무 : BOOL; (* AT %MW15.9 *)
    HMI_M_차종수정_차종_OPT1_VAN_유 : BOOL; (* AT %MW15.8 *)
    HMI_M_차종수정_차종_OPT1_슬라이딩_무 : BOOL; (* AT %MW15.1 *)
    HMI_M_차종수정_차종_OPT1_슬라이딩_유 : BOOL; (* AT %MW15.0 *)
    HMI_M_차종수정_차종_OPT1_폴딩_무 : BOOL; (* AT %MW15.5 *)
    HMI_M_차종수정_차종_OPT1_폴딩_유 : BOOL; (* AT %MW15.4 *)
    HMI_M_차종수정_차종_공대차 : BOOL; (* AT %MW20.12 *)
    HMI_M_차종수정_차종_공차 : BOOL; (* AT %MW20.10 *)
    HMI_M_차종수정_차종_불량대차 : BOOL; (* AT %MW20.13 *)
    HMI_M_차종수정_차종_불량차 : BOOL; (* AT %MW20.11 *)
    HMI_M_차종수정가능_OK : BOOL; (* AT %MW9.4 *)
    HMI_M_차종수정가능_SEL : BOOL; (* AT %MW9.3 *)
    HMI_M_현재표출_차종 : ARRAY[0..19] OF WORD; (* AT %MW30 *)
    HMI_차종매칭_공정선택 : WORD; (* AT %MW8 *)
    HMI_차종수정_공정선택 : WORD; (* AT %MW7 *)
    S101_M_자동_모드 : BOOL; (* AT %MW1000.1 *)
    S101_M_자동_운전중 : BOOL; (* AT %MW1000.4 *)
    S102_M_자동_모드 : BOOL; (* AT %MW1500.1 *)
    S103_M_자동_모드 : BOOL; (* AT %MW2000.1 *)
END_VAR
VAR
    HMI_BT_MODIFY : FB470_HMI_BType_Modify_LS;
END_VAR
VAR
    _t1 : BOOL;
    _t2 : BOOL;
    _p3 : BOOL;
    _t4 : BOOL;
    _t5 : BOOL;
    _e6 : F_TRIG;
    _e7 : F_TRIG;
END_VAR

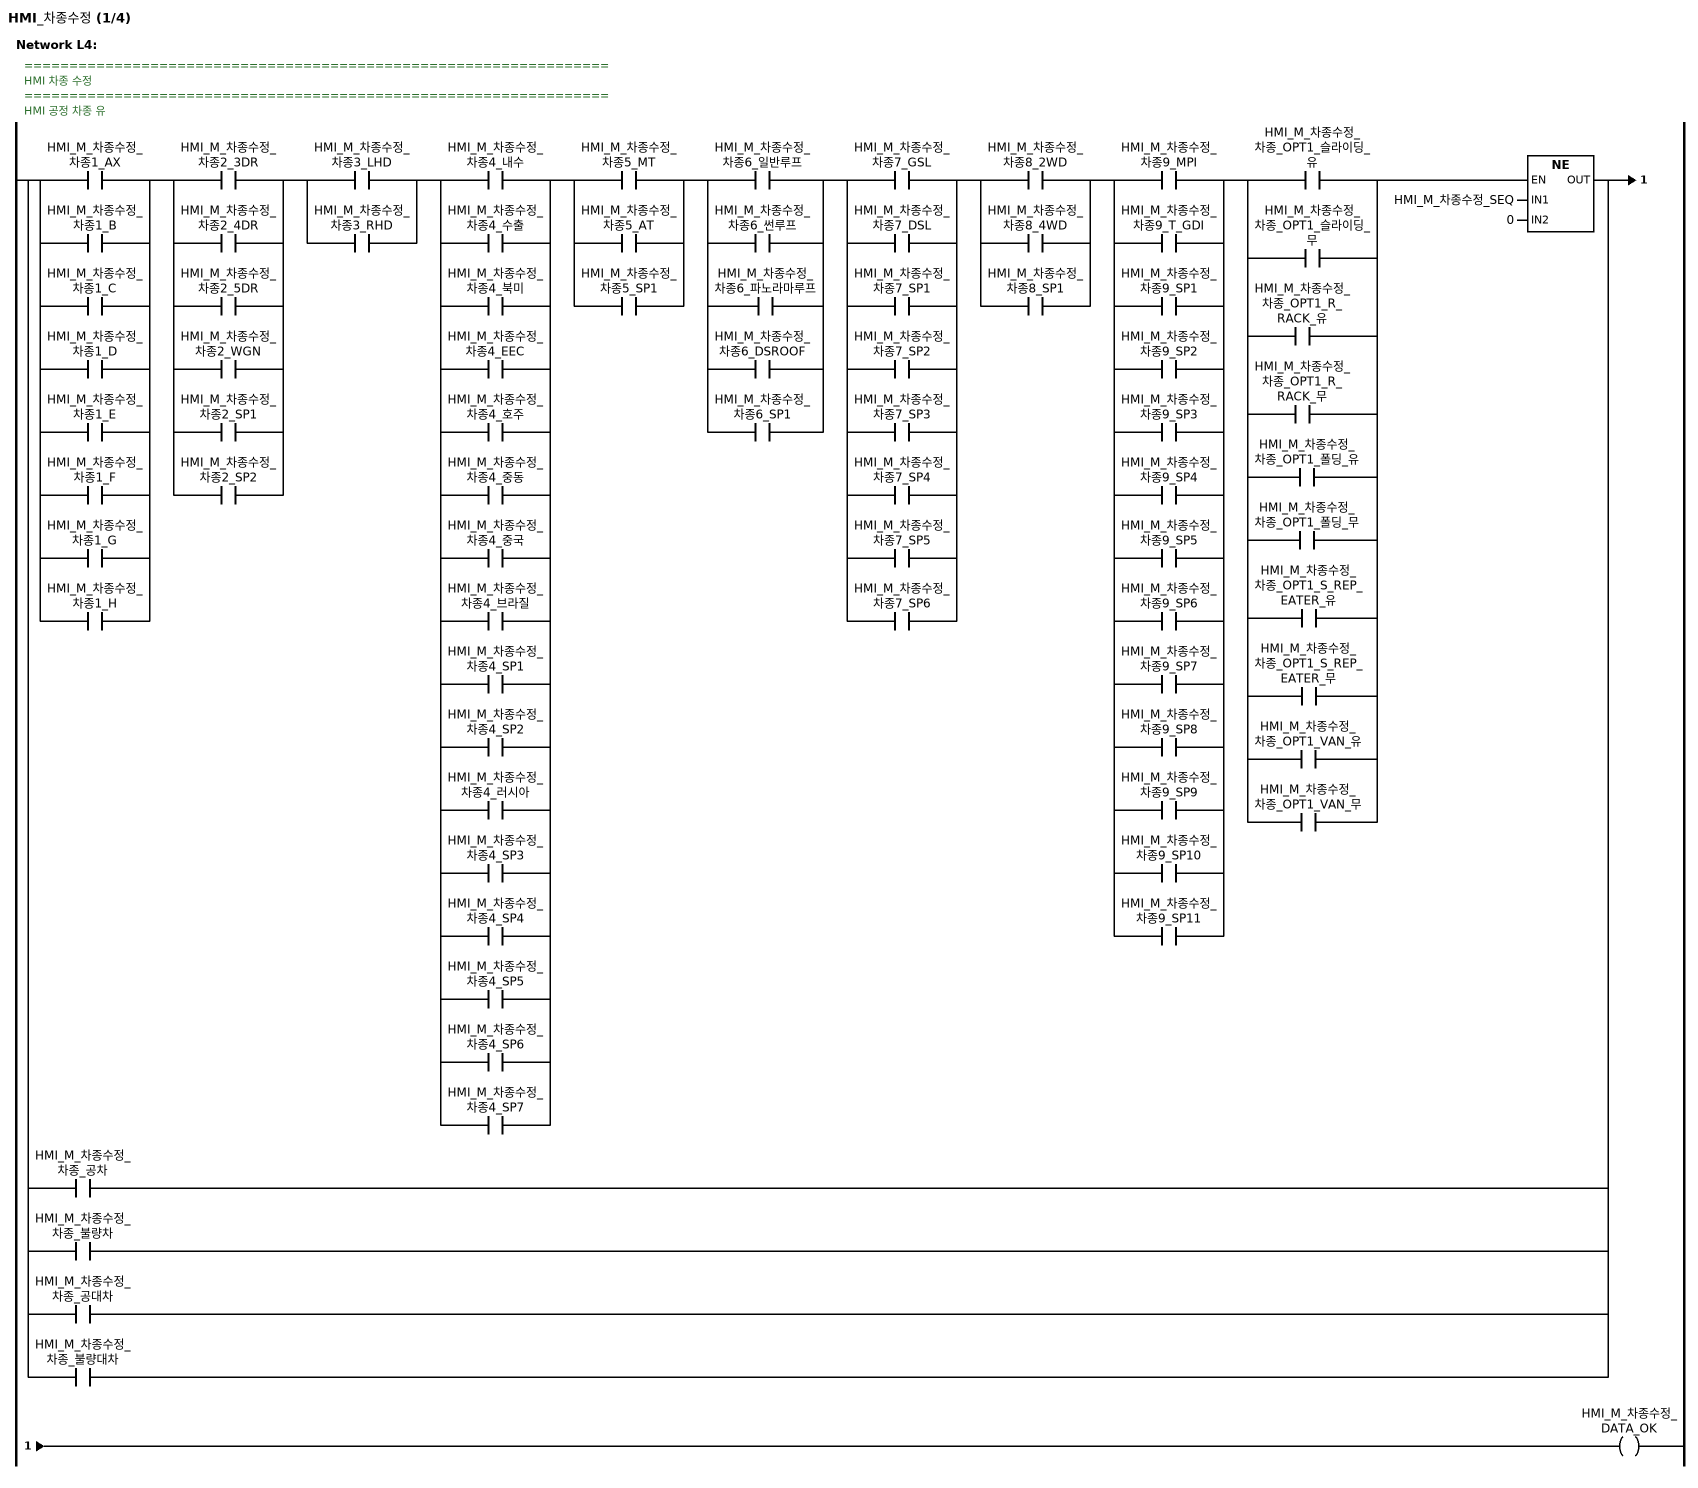
(* ================================================================= *)
(* HMI 차종 수정 *)
(* ================================================================= *)
(* HMI 공정 차종 유 *)
(* Rung L4 *)
IF (HMI_M_차종수정_차종1_AX OR HMI_M_차종수정_차종1_B OR HMI_M_차종수정_차종1_C OR HMI_M_차종수정_차종1_D OR HMI_M_차종수정_차종1_E OR HMI_M_차종수정_차종1_F OR HMI_M_차종수정_차종1_G OR HMI_M_차종수정_차종1_H) AND (HMI_M_차종수정_차종2_3DR OR HMI_M_차종수정_차종2_4DR OR HMI_M_차종수정_차종2_5DR OR HMI_M_차종수정_차종2_WGN OR HMI_M_차종수정_차종2_SP1 OR HMI_M_차종수정_차종2_SP2) AND (HMI_M_차종수정_차종3_LHD OR HMI_M_차종수정_차종3_RHD) AND (HMI_M_차종수정_차종4_내수 OR HMI_M_차종수정_차종4_수출 OR HMI_M_차종수정_차종4_북미 OR HMI_M_차종수정_차종4_EEC OR HMI_M_차종수정_차종4_호주 OR HMI_M_차종수정_차종4_중동 OR HMI_M_차종수정_차종4_중국 OR HMI_M_차종수정_차종4_브라질 OR HMI_M_차종수정_차종4_SP1 OR HMI_M_차종수정_차종4_SP2 OR HMI_M_차종수정_차종4_러시아 OR HMI_M_차종수정_차종4_SP3 OR HMI_M_차종수정_차종4_SP4 OR HMI_M_차종수정_차종4_SP5 OR HMI_M_차종수정_차종4_SP6 OR HMI_M_차종수정_차종4_SP7) AND (HMI_M_차종수정_차종5_MT OR HMI_M_차종수정_차종5_AT OR HMI_M_차종수정_차종5_SP1) AND (HMI_M_차종수정_차종6_일반루프 OR HMI_M_차종수정_차종6_썬루프 OR HMI_M_차종수정_차종6_파노라마루프 OR HMI_M_차종수정_차종6_DSROOF OR HMI_M_차종수정_차종6_SP1) AND (HMI_M_차종수정_차종7_GSL OR HMI_M_차종수정_차종7_DSL OR HMI_M_차종수정_차종7_SP1 OR HMI_M_차종수정_차종7_SP2 OR HMI_M_차종수정_차종7_SP3 OR HMI_M_차종수정_차종7_SP4 OR HMI_M_차종수정_차종7_SP5 OR HMI_M_차종수정_차종7_SP6) AND (HMI_M_차종수정_차종8_2WD OR HMI_M_차종수정_차종8_4WD OR HMI_M_차종수정_차종8_SP1) AND (HMI_M_차종수정_차종9_MPI OR HMI_M_차종수정_차종9_T_GDI OR HMI_M_차종수정_차종9_SP1 OR HMI_M_차종수정_차종9_SP2 OR HMI_M_차종수정_차종9_SP3 OR HMI_M_차종수정_차종9_SP4 OR HMI_M_차종수정_차종9_SP5 OR HMI_M_차종수정_차종9_SP6 OR HMI_M_차종수정_차종9_SP7 OR HMI_M_차종수정_차종9_SP8 OR HMI_M_차종수정_차종9_SP9 OR HMI_M_차종수정_차종9_SP10 OR HMI_M_차종수정_차종9_SP11) AND (HMI_M_차종수정_차종_OPT1_슬라이딩_유 OR HMI_M_차종수정_차종_OPT1_슬라이딩_무 OR HMI_M_차종수정_차종_OPT1_R_RACK_유 OR HMI_M_차종수정_차종_OPT1_R_RACK_무 OR HMI_M_차종수정_차종_OPT1_폴딩_유 OR HMI_M_차종수정_차종_OPT1_폴딩_무 OR HMI_M_차종수정_차종_OPT1_S_REP_EATER_유 OR HMI_M_차종수정_차종_OPT1_S_REP_EATER_무 OR HMI_M_차종수정_차종_OPT1_VAN_유 OR HMI_M_차종수정_차종_OPT1_VAN_무) THEN
    _t1 := HMI_M_차종수정_SEQ <> 0;
END_IF;
HMI_M_차종수정_DATA_OK := _t1 OR HMI_M_차종수정_차종_공차 OR HMI_M_차종수정_차종_불량차 OR HMI_M_차종수정_차종_공대차 OR HMI_M_차종수정_차종_불량대차;

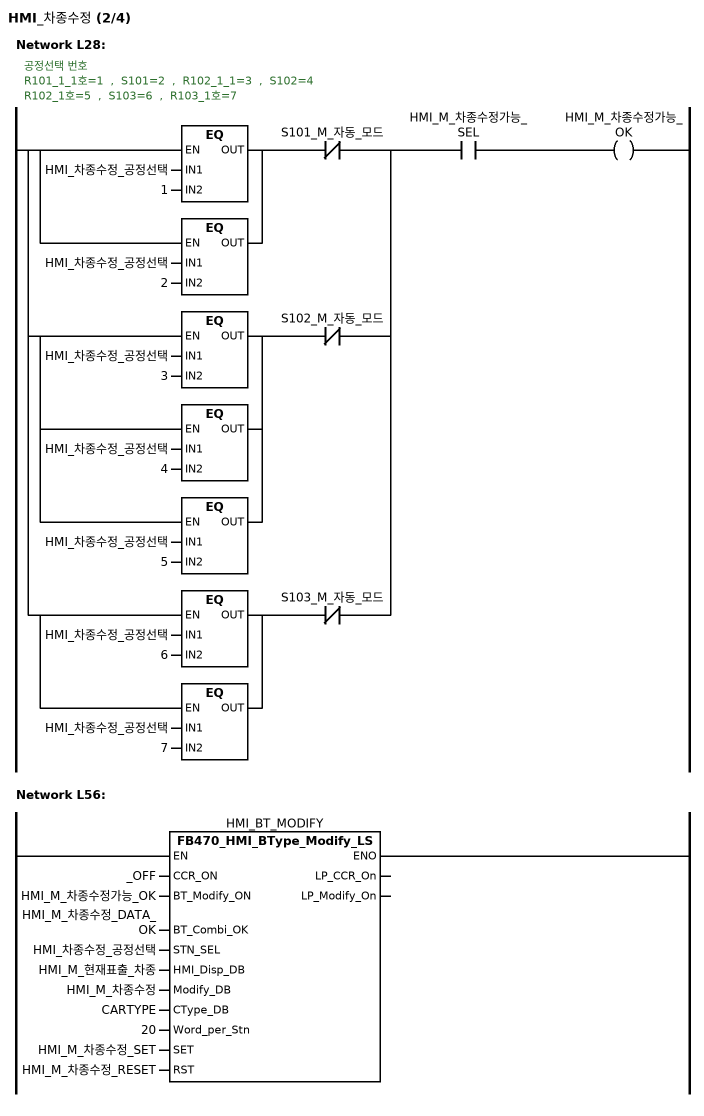
(* 공정선택 번호 *)
(* R101_1_1호=1  ,  S101=2  ,  R102_1_1=3  ,  S102=4 *)
(* R102_1호=5  ,  S103=6  ,  R103_1호=7 *)
(* Rung L28 *)
HMI_M_차종수정가능_OK := ((((HMI_차종수정_공정선택 = 1) OR (HMI_차종수정_공정선택 = 2)) AND NOT S101_M_자동_모드) OR (((HMI_차종수정_공정선택 = 3) OR (HMI_차종수정_공정선택 = 4) OR (HMI_차종수정_공정선택 = 5)) AND NOT S102_M_자동_모드) OR (((HMI_차종수정_공정선택 = 6) OR (HMI_차종수정_공정선택 = 7)) AND NOT S103_M_자동_모드)) AND HMI_M_차종수정가능_SEL;
(* Rung L56 *)
HMI_BT_MODIFY(CCR_ON := _OFF, BT_Modify_ON := HMI_M_차종수정가능_OK, BT_Combi_OK := HMI_M_차종수정_DATA_OK, STN_SEL := HMI_차종수정_공정선택, HMI_Disp_DB := HMI_M_현재표출_차종, Modify_DB := HMI_M_차종수정, CType_DB := CARTYPE, Word_per_Stn := 20, SET := HMI_M_차종수정_SET, RST := HMI_M_차종수정_RESET);

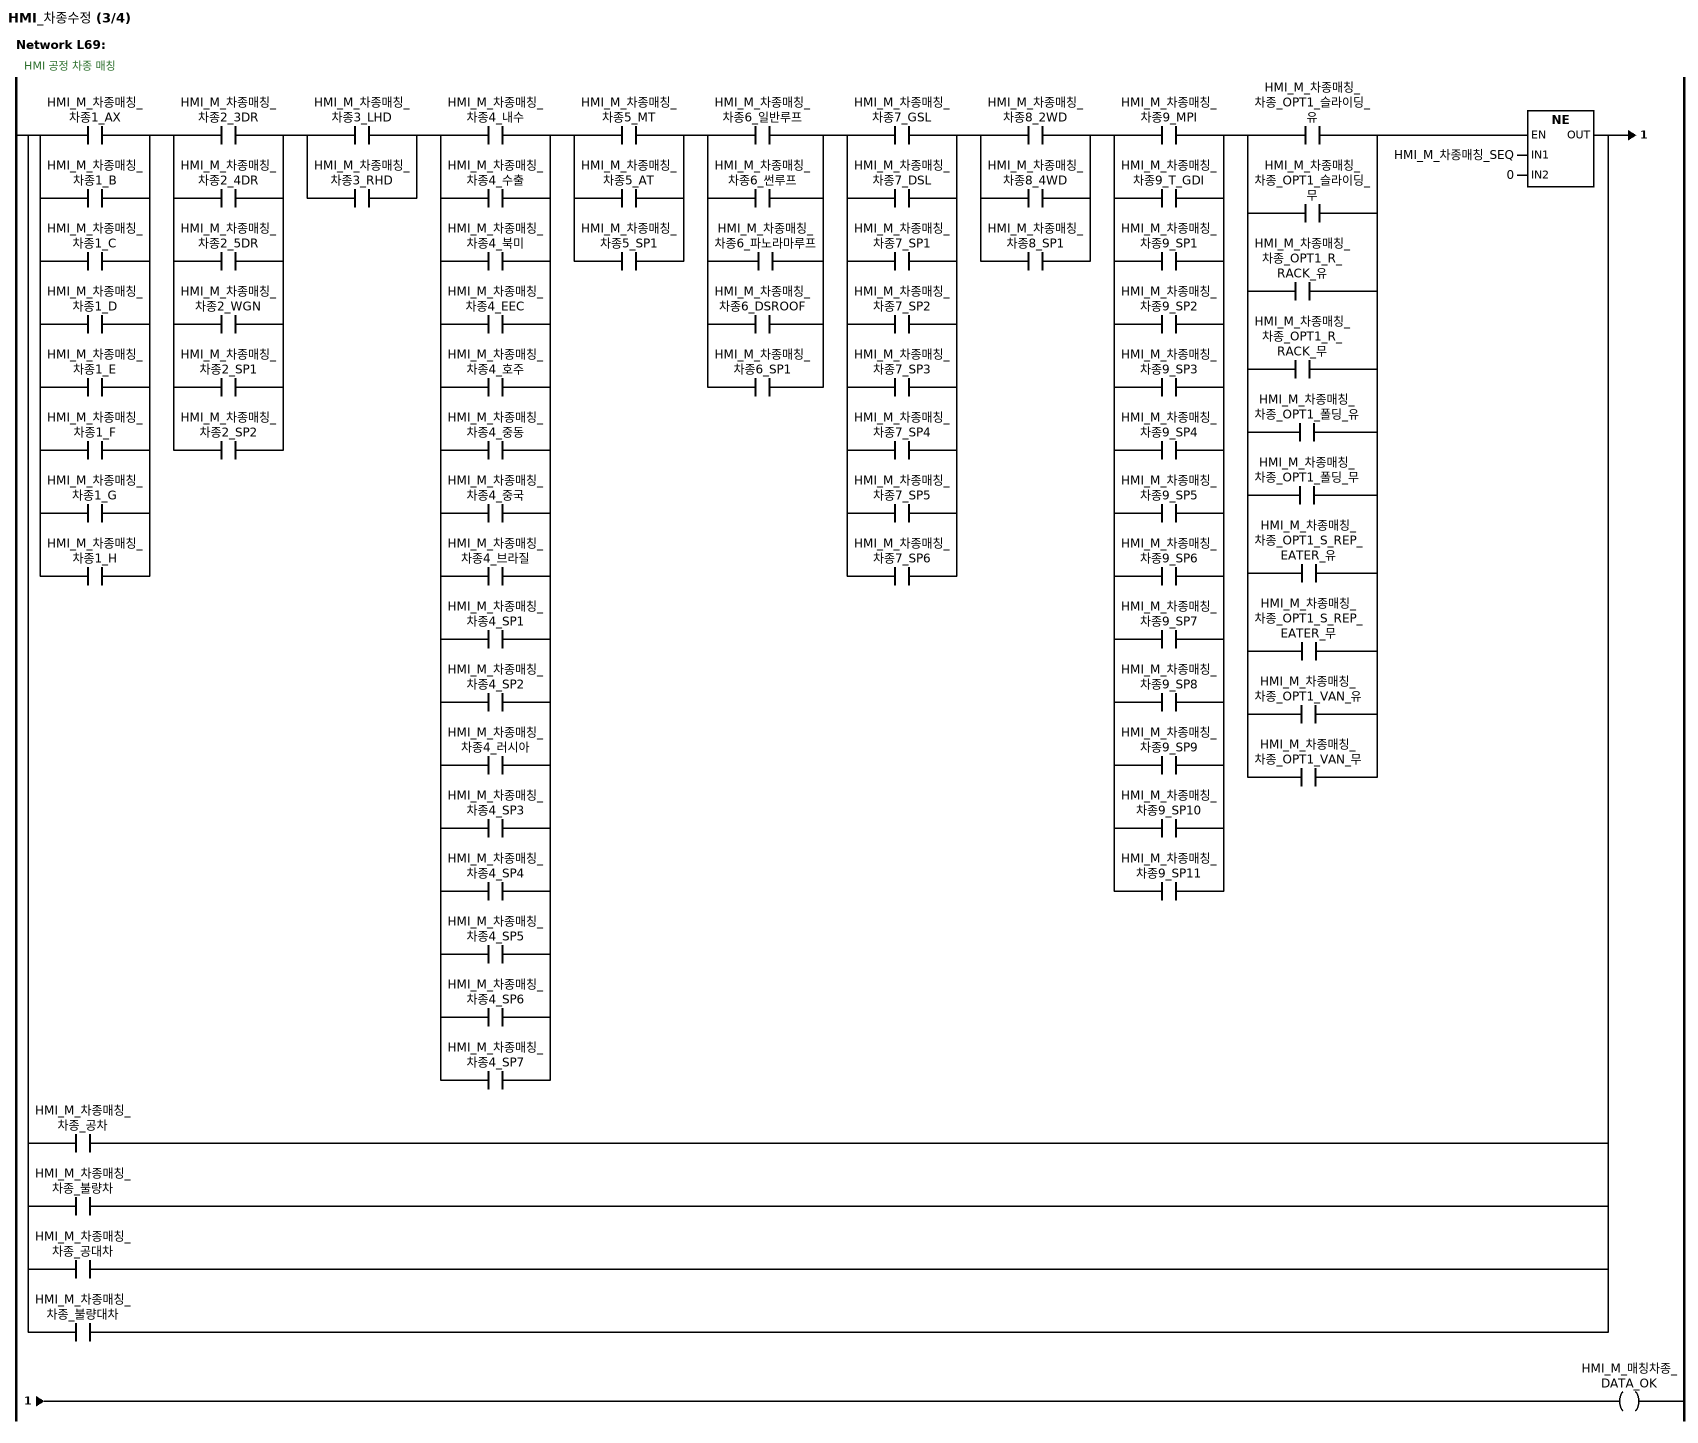
(* HMI 공정 차종 매칭 *)
(* Rung L69 *)
IF (HMI_M_차종매칭_차종1_AX OR HMI_M_차종매칭_차종1_B OR HMI_M_차종매칭_차종1_C OR HMI_M_차종매칭_차종1_D OR HMI_M_차종매칭_차종1_E OR HMI_M_차종매칭_차종1_F OR HMI_M_차종매칭_차종1_G OR HMI_M_차종매칭_차종1_H) AND (HMI_M_차종매칭_차종2_3DR OR HMI_M_차종매칭_차종2_4DR OR HMI_M_차종매칭_차종2_5DR OR HMI_M_차종매칭_차종2_WGN OR HMI_M_차종매칭_차종2_SP1 OR HMI_M_차종매칭_차종2_SP2) AND (HMI_M_차종매칭_차종3_LHD OR HMI_M_차종매칭_차종3_RHD) AND (HMI_M_차종매칭_차종4_내수 OR HMI_M_차종매칭_차종4_수출 OR HMI_M_차종매칭_차종4_북미 OR HMI_M_차종매칭_차종4_EEC OR HMI_M_차종매칭_차종4_호주 OR HMI_M_차종매칭_차종4_중동 OR HMI_M_차종매칭_차종4_중국 OR HMI_M_차종매칭_차종4_브라질 OR HMI_M_차종매칭_차종4_SP1 OR HMI_M_차종매칭_차종4_SP2 OR HMI_M_차종매칭_차종4_러시아 OR HMI_M_차종매칭_차종4_SP3 OR HMI_M_차종매칭_차종4_SP4 OR HMI_M_차종매칭_차종4_SP5 OR HMI_M_차종매칭_차종4_SP6 OR HMI_M_차종매칭_차종4_SP7) AND (HMI_M_차종매칭_차종5_MT OR HMI_M_차종매칭_차종5_AT OR HMI_M_차종매칭_차종5_SP1) AND (HMI_M_차종매칭_차종6_일반루프 OR HMI_M_차종매칭_차종6_썬루프 OR HMI_M_차종매칭_차종6_파노라마루프 OR HMI_M_차종매칭_차종6_DSROOF OR HMI_M_차종매칭_차종6_SP1) AND (HMI_M_차종매칭_차종7_GSL OR HMI_M_차종매칭_차종7_DSL OR HMI_M_차종매칭_차종7_SP1 OR HMI_M_차종매칭_차종7_SP2 OR HMI_M_차종매칭_차종7_SP3 OR HMI_M_차종매칭_차종7_SP4 OR HMI_M_차종매칭_차종7_SP5 OR HMI_M_차종매칭_차종7_SP6) AND (HMI_M_차종매칭_차종8_2WD OR HMI_M_차종매칭_차종8_4WD OR HMI_M_차종매칭_차종8_SP1) AND (HMI_M_차종매칭_차종9_MPI OR HMI_M_차종매칭_차종9_T_GDI OR HMI_M_차종매칭_차종9_SP1 OR HMI_M_차종매칭_차종9_SP2 OR HMI_M_차종매칭_차종9_SP3 OR HMI_M_차종매칭_차종9_SP4 OR HMI_M_차종매칭_차종9_SP5 OR HMI_M_차종매칭_차종9_SP6 OR HMI_M_차종매칭_차종9_SP7 OR HMI_M_차종매칭_차종9_SP8 OR HMI_M_차종매칭_차종9_SP9 OR HMI_M_차종매칭_차종9_SP10 OR HMI_M_차종매칭_차종9_SP11) AND (HMI_M_차종매칭_차종_OPT1_슬라이딩_유 OR HMI_M_차종매칭_차종_OPT1_슬라이딩_무 OR HMI_M_차종매칭_차종_OPT1_R_RACK_유 OR HMI_M_차종매칭_차종_OPT1_R_RACK_무 OR HMI_M_차종매칭_차종_OPT1_폴딩_유 OR HMI_M_차종매칭_차종_OPT1_폴딩_무 OR HMI_M_차종매칭_차종_OPT1_S_REP_EATER_유 OR HMI_M_차종매칭_차종_OPT1_S_REP_EATER_무 OR HMI_M_차종매칭_차종_OPT1_VAN_유 OR HMI_M_차종매칭_차종_OPT1_VAN_무) THEN
    _t2 := HMI_M_차종매칭_SEQ <> 0;
END_IF;
HMI_M_매칭차종_DATA_OK := _t2 OR HMI_M_차종매칭_차종_공차 OR HMI_M_차종매칭_차종_불량차 OR HMI_M_차종매칭_차종_공대차 OR HMI_M_차종매칭_차종_불량대차;

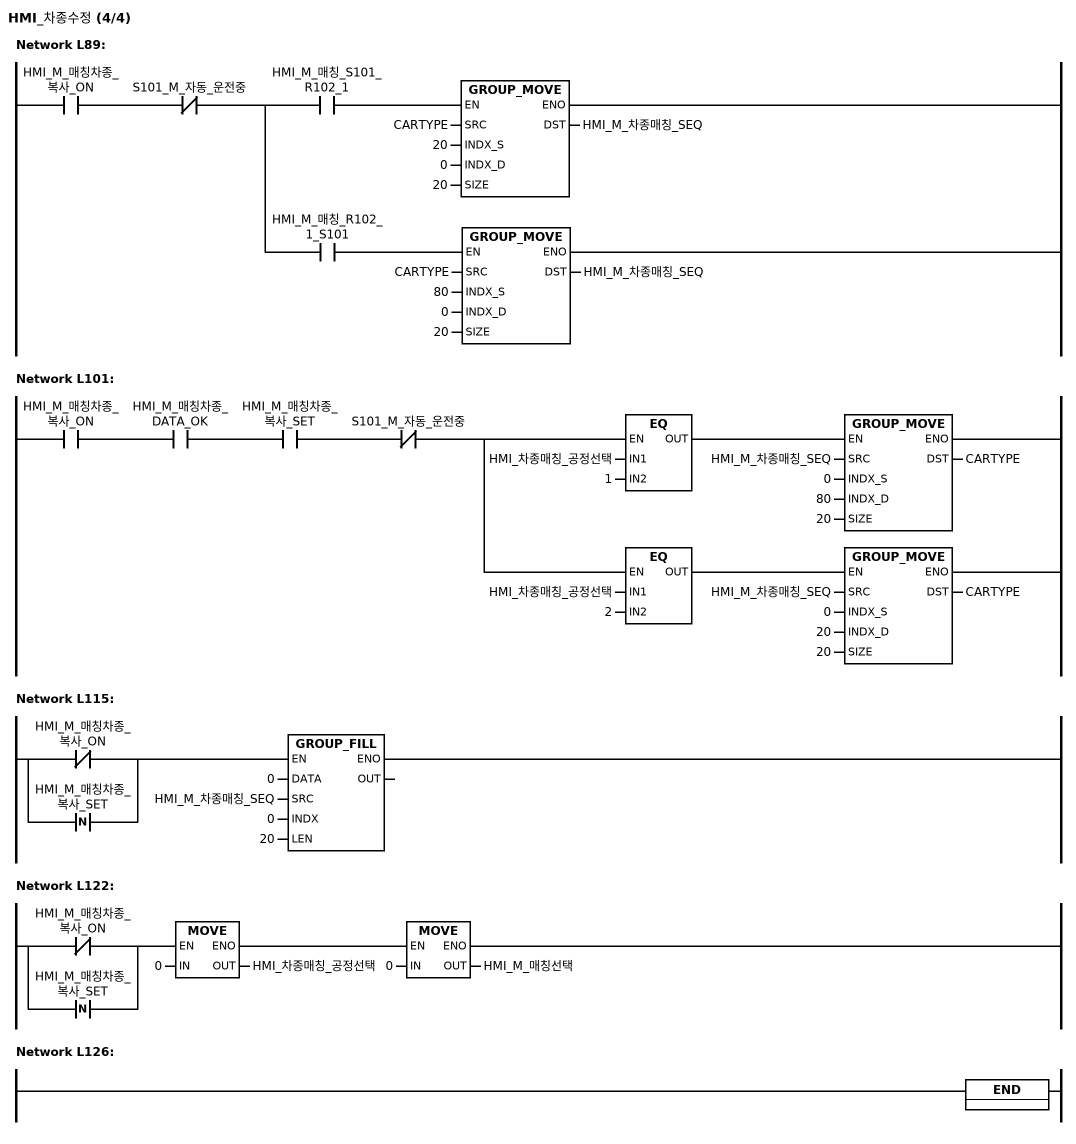
(* Rung L89 *)
IF HMI_M_매칭차종_복사_ON AND NOT S101_M_자동_운전중 AND HMI_M_매칭_S101_R102_1 THEN
    HMI_M_차종매칭_SEQ := GROUP_MOVE(SRC := CARTYPE, INDX_S := 20, INDX_D := 0, SIZE := 20);
END_IF;
IF HMI_M_매칭차종_복사_ON AND NOT S101_M_자동_운전중 AND HMI_M_매칭_R102_1_S101 THEN
    HMI_M_차종매칭_SEQ := GROUP_MOVE(SRC := CARTYPE, INDX_S := 80, INDX_D := 0, SIZE := 20);
END_IF;
(* Rung L101 *)
_p3 := HMI_M_매칭차종_복사_ON AND HMI_M_매칭차종_DATA_OK AND HMI_M_매칭차종_복사_SET AND NOT S101_M_자동_운전중;
IF _p3 THEN _t4 := HMI_차종매칭_공정선택 = 1; END_IF;
IF _t4 THEN CARTYPE := GROUP_MOVE(SRC := HMI_M_차종매칭_SEQ, INDX_S := 0, INDX_D := 80, SIZE := 20); END_IF;
IF _p3 THEN _t5 := HMI_차종매칭_공정선택 = 2; END_IF;
IF _t5 THEN CARTYPE := GROUP_MOVE(SRC := HMI_M_차종매칭_SEQ, INDX_S := 0, INDX_D := 20, SIZE := 20); END_IF;
(* Rung L115 *)
_e6(CLK := HMI_M_매칭차종_복사_SET);
IF NOT HMI_M_매칭차종_복사_ON OR _e6.Q THEN
    GROUP_FILL(DATA := 0, SRC := HMI_M_차종매칭_SEQ, INDX := 0, LEN := 20);
END_IF;
(* Rung L122 *)
_e7(CLK := HMI_M_매칭차종_복사_SET);
IF NOT HMI_M_매칭차종_복사_ON OR _e7.Q THEN
    HMI_차종매칭_공정선택 := 0;
    HMI_M_매칭선택 := 0;
END_IF;
(* Rung L126 *)
END();
END_PROGRAM

PROGRAM 알람트래킹 (* task: 스캔 프로그램 *)

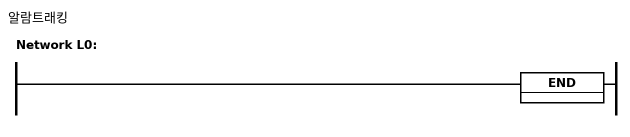
(* Rung L0 *)
END();
END_PROGRAM